{attribute 'linkalways'} 
{attribute 'no_explicit_call' := 'This FB is a CLASS and must be accessed using methods or properties'}
{attribute 'enable_dynamic_creation'}
FUNCTION_BLOCK _ETcVnDistanceType EXTENDS EnumDatatypeBase
VAR
	localData : ETcVnDistanceType;
	activeData : REFERENCE TO ETcVnDistanceType;
	enumBaseDatatype : _DINT(localData);
END_VAR

METHOD PRIVATE AddLocalEnumeration
VAR_INPUT
	Enumeration : T_MAXSTRING;
	Value : ETcVnDistanceType;
END_VAR
AddEnumeration(Enumeration, Value);
END_METHOD

PROPERTY PUBLIC Address : PVOID
GET
Address := ADR(activeData);
END_GET
END_PROPERTY

METHOD PUBLIC ClearReference
VAR_INPUT
END_VAR
activeData REF= localData;
SetBaseDatatypeReference();
END_METHOD

METHOD PUBLIC Clone : I_Datatype
VAR
    pClone : POINTER TO _ETcVnDistanceType;
END_VAR
pClone := __NEW(_ETcVnDistanceType(InitialValue := Value));
Clone := pClone^;
END_METHOD

METHOD FB_init : BOOL
VAR_INPUT
	bInitRetains : BOOL; // if TRUE, the retain variables are initialized (warm start / cold start)
	bInCopyCode : BOOL;  // if TRUE, the instance afterwards gets moved into the copy code (online change)
	InitialValue : ETcVnDistanceType;
END_VAR
localData := InitialValue;
AddBaseDatatype(enumBaseDatatype);
ClearReference();

AddLocalEnumeration('TCVN_DT_USER', ETcVnDistanceType.TCVN_DT_USER);
AddLocalEnumeration('TCVN_DT_L1', ETcVnDistanceType.TCVN_DT_L1);
AddLocalEnumeration('TCVN_DT_L2', ETcVnDistanceType.TCVN_DT_L2);
AddLocalEnumeration('TCVN_DT_C', ETcVnDistanceType.TCVN_DT_C);
AddLocalEnumeration('TCVN_DT_L12', ETcVnDistanceType.TCVN_DT_L12);
AddLocalEnumeration('TCVN_DT_FAIR', ETcVnDistanceType.TCVN_DT_FAIR);
AddLocalEnumeration('TCVN_DT_WELSCH', ETcVnDistanceType.TCVN_DT_WELSCH);
AddLocalEnumeration('TCVN_DT_HUBER ', ETcVnDistanceType.TCVN_DT_HUBER);
END_METHOD

PROPERTY PUBLIC Identifier : T_MAXSTRING
GET
Identifier := 'ETcVnDistanceType';
END_GET
END_PROPERTY

METHOD IsEnumeratorValueEqual : BOOL
VAR_INPUT
	Enumerator : I_KeyValueForwardEnumerator;
END_VAR
VAR
	storedValue : ETcVnDistanceType;
END_VAR
IF NOT Enumerator.TryGet(storedValue) THEN
	RETURN;
END_IF

IsEnumeratorValueEqual := storedValue = activeData;
END_METHOD

METHOD PUBLIC MakeReferenceTo
VAR_INPUT
	ReferenceTarget : REFERENCE TO ETcVnDistanceType;
END_VAR
activeData REF= ReferenceTarget;
SetBaseDatatypeReference();
END_METHOD

METHOD PROTECTED SetBaseDatatypeReference
VAR_INPUT
END_VAR
enumBaseDatatype.MakeReferenceTo(activeData);
END_METHOD

PROPERTY PUBLIC Size : UDINT
GET
Size := SIZEOF(activeData);
END_GET
END_PROPERTY

METHOD TryMakeReferenceTo : BOOL
VAR_INPUT
	Target : I_Datatype;
END_VAR
VAR
	targetAsEnum : I_EnumDatatype;
	pTargetData : POINTER TO ETcVnDistanceType;
END_VAR
IF NOT Target.TryResolveAsEnumDatatype(targetAsEnum) THEN
	RETURN;
END_IF

IF targetAsEnum.Identifier <> Identifier THEN
	RETURN;
END_IF

pTargetData := Target.Address;
activeData REF= pTargetData^;
SetBaseDatatypeReference();
TryMakeReferenceTo := TRUE;
END_METHOD

PROPERTY PUBLIC Value : ETcVnDistanceType
GET
Value := activeData;
END_GET
SET
activeData := Value;
END_SET
END_PROPERTY

END_FUNCTION_BLOCK

(* stored: Version 1.1.0.1, ProductVersion 3.1.4024.12
   POU _ETcVnDistanceType: Id {b444cd76-783b-4850-a3e5-3718c2b91fbe}, SpecialFunc None
   Folder Constructor: Id {da548066-eba5-40ea-adea-44fd18f60fb9}
   Folder Private: Id {62fb2e76-9053-4f95-9c3e-df3f518877af}
   Folder Protected: Id {3b011a3b-6aed-4b22-81d4-40dfbce3cc0d}
   Method AddLocalEnumeration: Id {13294c17-76ca-422a-b427-f91814689e4c}
   Property Address: Id {20a182fe-196e-4e80-8464-d814ff71de15}
   Get Get: Id {f3011c29-0632-475b-bde9-957360a7204c}
   Method ClearReference: Id {79db0e77-2839-43cd-94d0-4020c0bfe54c}
   Method Clone: Id {bbfba4f9-96ef-43c9-8e78-103634495783}
   Method FB_init: Id {cf57ec40-0a4a-4b84-beea-5ad21f19ac9c}
   Property Identifier: Id {5acb8cd7-e1cc-4cbb-8e65-93fb11660278}
   Get Get: Id {635f770a-0989-4ff3-8ad7-4098c0e5d883}
   Method IsEnumeratorValueEqual: Id {5d448bc5-5c62-4012-a6e6-9e6bdd4f5e7c}
   Method MakeReferenceTo: Id {33fcb602-a637-4ada-846f-d25621f6e17d}
   Method SetBaseDatatypeReference: Id {0caf90e0-e8ba-4742-87e2-dc0f4169e1dc}
   Property Size: Id {50bf3e4c-6c9b-4bc3-be74-481eb77f94f7}
   Get Get: Id {a29434a0-560a-49b3-a42a-0f1d52ca5250}
   Method TryMakeReferenceTo: Id {648d6f13-1138-4e47-89de-2021b2c90753}
   Property Value: Id {e66d7d51-86ec-4913-82d7-ca61bdc2a6e6}
   Get Get: Id {b6e801a5-ad37-470e-92a4-92051afd7338}
   Set Set: Id {1bdfd23e-a30e-4081-a127-be9f5b84ead0} *)
